// Mitsubishi GX Works2 project: PGC(shorter)   PLC: FX1N/FX1NC

PROGRAM MAIN
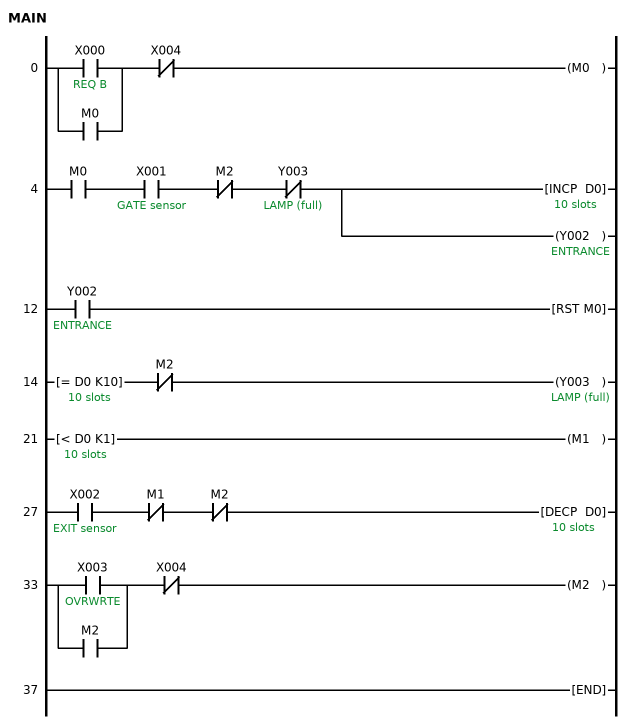
0     LD      X000  ; REQ B
      OR      M0
      ANI     X004
      OUT     M0
4     LD      M0
      AND     X001  ; GATE sensor
      ANI     M2
      ANI     Y003  ; LAMP (full)
      INCP    D0  ; 10 slots
      OUT     Y002  ; ENTRANCE
12    LD      Y002  ; ENTRANCE
      RST     M0
14    LD=     D0 K10  ; 10 slots
      ANI     M2
      OUT     Y003  ; LAMP (full)
21    LD<     D0 K1  ; 10 slots
      OUT     M1
27    LD      X002  ; EXIT sensor
      ANI     M1
      ANI     M2
      DECP    D0
33    LD      X003  ; OVRWRTE
      OR      M2
      ANI     X004
      OUT     M2
37    END
END_PROGRAM
